{attribute 'qualified_only'}
{attribute 'strict'}
{attribute 'to_string'}
TYPE eNetContactorState :
(
	Open 			:= 0,
	RightClosed		:= 1,
	LeftClosed		:= 2
);
END_TYPE

(* stored: Version 1.1.0.1, ProductVersion 3.1.4026.18
   DUT eNetContactorState: Id {400ec5f5-6a51-45d4-ab89-88d41061802c} *)
